// Block: AreaXX_FinalCutLub_PERS

DATA_BLOCK AreaXX_FinalCutLub_PERS
VERSION : 0.1
   NON_RETAIN
   VAR
      PersistentValues : Struct
         Data : Struct
            SavedCutBenchCode : DInt;
            PumpJobCounter : UDInt;
            JobsCounter : UDInt;
         END_STRUCT;
         Par : Struct
            SystemOffOn : Bool;
            JobsToStart : UDInt;
            OilPumpCycles : UDInt;
         END_STRUCT;
      END_STRUCT;
   END_VAR

BEGIN
   // No initialization required
END_DATA_BLOCK
